Staubli VAL3: JPOINT.dtx

public string sItems
string sPathTemplate = "Disk://kernel/template/JPOINT"
public bool bMoveType[3]
public bool bStepping
pointRx pToGo = {fatherId=world[0]}
pointRx pLastPoint = {fatherId=world[0]}
mdesc nom_speed = {accel=50, vel=50, decel=50, blend=off}
num nTcpAction
pointRx pPointTo = {fatherId=world[0]}
string sTrajType
string sMenu[8]
mdesc mMdesc = {accel=25, vel=25, decel=25, blend=off}
bool bToSave
InstrItem tcpInstr
  [0]
    string sType
    string sData
public Trajectory tTraj
  [0]
    TrajectoryItem tSuper
      [0]
        num distance
        num moveType
        num nTime
        num nStop
        num nTcpAction
        string comment
        bool toStop
        mdesc nom_speed = {tmax=300, rmax=9999, leave=30, reach=30}
        InstrItem iInstr[3]
          [0]
            string sType
            string sData
          [1]
            string sType
            string sData
          [2]
            string sType
            string sData
        num nMoveId
    string sID
    num nId
num nIndex
num nKey
TrajJoint jEditPoint
  [0]
    num nIndexTool
    TrajJointItem tData
      [0]
        jointRx jJoint
        TrajectoryItem tSuper
          [0]
            num distance
            num moveType
            num nTime
            num nStop
            num nTcpAction
            string comment
            bool toStop
            mdesc nom_speed = {tmax=9999, rmax=9999, leave=30, reach=30}
            InstrItem iInstr[3]
              [0]
                string sType
                string sData
              [1]
                string sType
                string sData
              [2]
                string sType
                string sData
            num nMoveId
    string sID
    num nIndexFrame
string sTrajCycle
